VISUALIZATION Infoseite  // 800x480
END_VISUALIZATION

(* stored: Version 1.1.0.1, ProductVersion 3.1.4022.6
   Visu Infoseite: Id {4d7a476a-6aa8-40a7-8fbe-f8e9c80665f1} *)
